PROGRAM Alarming
VAR
	bInit	: BOOL := TRUE;
	bSend	: BOOL;

	fbMsg	: FB_TcMessage;
END_VAR

IF bInit THEN
	bInit := FALSE;
	fbMsg.CreateEx(TC_EVENTS.MyEventClass.MyFirstMessage, 0);
END_IF

IF bSend THEN
	bSend := FALSE;
	fbMsg.Send(0);
END_IF

END_PROGRAM

(* stored: Version 1.1.0.1, ProductVersion 3.1.4024.12
   POU Alarming: Id {badb9cdc-1cfe-457d-b1ef-bbaeee5672aa}, SpecialFunc None *)
